Staubli VAL3: setTool.pgx

public program setTool(num nTool (dimensions=1))
begin
  switch nTool
    case 0
      tActive=flange
    break
    case 1
      tActive=tGripper
    break
    case 2
    break
    default
      logMsg("erro setTool: "+chr(nTool))
    break
  endSwitch
end
